// TIA Portal project "2020-11-13_LampeggioMacchinaStati" (V16)
// Programma che gestisce la ventilazione di un motore

(* hardware
DEVICE "Stazione SIMATIC 1200_1"  S71200.Device
   slot 0: "Telaio di montaggio S7-1200"  Rack  V1.0
   slot 1: "PLC_1"  CPU 1215C DC/DC/DC  6ES7 215-1AG40-0XB0  V4.2
*)

// ===== PLC "PLC_1"  CPU 1215C DC/DC/DC =====

VAR_GLOBAL   // PLC tag table "Tabella delle variabili standard"
   "in0_f" AT %I0.0 : Bool;
   "in1_f" AT %I0.1 : Bool;
   "in2_f" AT %I0.2 : Bool;
   "in3_f" AT %I0.3 : Bool;
   "in4_f" AT %I0.4 : Bool;
   "in5_f" AT %I0.5 : Bool;
   "in6_f" AT %I0.6 : Bool;
   "out0" AT %Q0.0 : Bool;
   "out1" AT %Q0.1 : Bool;
   "in7_f" AT %I0.7 : Bool;
   "out2" AT %Q0.2 : Bool;
   "out3" AT %Q0.3 : Bool;
   "out4" AT %Q0.4 : Bool;
   "sempre vero" AT %M7.0 : Bool;   // bit sempre vero
   "uscite byte" AT %QB0 : Byte;   // Uscite fisiche
   "uscite memorie" AT %MB1 : Byte;   // uscite memorie da usare come ingressi
   "out4_M" AT %M1.4 : Bool;
   "out3_M" AT %M1.3 : Bool;
   "out2_M" AT %M1.2 : Bool;
   "out1_M" AT %M1.1 : Bool;
   "out0_M" AT %M1.0 : Bool;
   "ingressi byte" AT %IB0 : Byte;   // Ingressi fisici
   "ingressi memorie" AT %MB0 : Byte;   // Ingressi Na non filtrati
   "in0_na" AT %M0.0 : Bool;
   "in1_na" AT %M0.1 : Bool;
   "in2_na" AT %M0.2 : Bool;
   "in3_na" AT %M0.3 : Bool;
   "in4_na" AT %M0.4 : Bool;
   "in5_na" AT %M0.5 : Bool;
   "in6_na" AT %M0.6 : Bool;
   "in7_na" AT %M0.7 : Bool;
   "out5" AT %Q0.5 : Bool;
   "out6" AT %Q0.6 : Bool;
   "out7" AT %Q0.7 : Bool;
   "out5_M" AT %M1.5 : Bool;
   "out6_M" AT %M1.6 : Bool;
   "out7_M" AT %M1.7 : Bool;
   "ingressi memorie filtrato" AT %MB2 : Byte;
   "in0" AT %M2.0 : Bool;
   "in1" AT %M2.1 : Bool;
   "in2" AT %M2.2 : Bool;
   "in3" AT %M2.3 : Bool;
   "in4" AT %M2.4 : Bool;
   "in5" AT %M2.5 : Bool;
   "in6" AT %M2.6 : Bool;
   "in7" AT %M2.7 : Bool;
   "ingressi memorie_p" AT %MB3 : Byte;
   "in0_p" AT %M3.0 : Bool;   // finecorsa di sicurezza
   "in1_p" AT %M3.1 : Bool;   // presenza tensione al motore
   "in2_p" AT %M3.2 : Bool;   // presenza Allarme
   "in3_p" AT %M3.3 : Bool;   // ventilazione motore ON
   "in4_p" AT %M3.4 : Bool;   // motore troppo caldo
   "in5_p" AT %M3.5 : Bool;   // comando avviamento motore
   "in6_p" AT %M3.6 : Bool;   // comando arresto motore
   "in7_p" AT %M3.7 : Bool;   // Reset memorizzazione Allarme
   "ingressi_memorie_var_p" AT %MB4 : Byte;
   "in0_var_p" AT %M4.0 : Bool;   // finecorsa di sicurezza
   "in1_var_p" AT %M4.1 : Bool;   // presenza tensione al motore
   "in2_var_p" AT %M4.2 : Bool;   // presenza Allarme
   "in3_var_p" AT %M4.3 : Bool;   // ventilazione motore ON
   "in4_var_p" AT %M4.4 : Bool;   // motore troppo caldo
   "in5_var_p" AT %M4.5 : Bool;   // comando avviamento motore
   "in6_var_p" AT %M4.6 : Bool;   // comando arresto motore
   "in7_var_p" AT %M4.7 : Bool;   // Reset memorizzazione Allarme
   "Stato" AT %MB8 : Byte;
   "Stato_futuro" AT %MB9 : Byte;
   "Stato_old" AT %MB10 : Byte;
END_VAR

VAR_GLOBAL CONSTANT   // PLC tag table "Tabella delle variabili standard"
   "maschera NCNA" : Byte := B#2#00000000;   // mettere a 1 i bit NC
   "filtro in0" : Time := T#500ms;
   "filtro in1" : Time := T#100ms;
   "filtro in2" : Time := T#100ms;
   "filtro in3" : Time := T#100ms;
   "filtro in4" : Time := T#100ms;
   "filtro in5" : Time := T#100ms;
   "filtro in6" : Time := T#100ms;
   "filtro in7" : Time := T#100ms;
   "Maschera Out Reset" : Byte := B#2#00000000;
   "Stato_partenza" : Byte := 0;
END_VAR

// folder: System blocks/Program resources

DATA_BLOCK "filtro_in0"   // DB1
{ S7_Optimized_Access := 'TRUE' }
AUTHOR : Simatic
FAMILY : IEC
NAME : IEC_TMR
VERSION : 1.0
// stored: InstanceOfName IEC_TIMER
"IEC_TIMER"
BEGIN
END_DATA_BLOCK

DATA_BLOCK "filtro_in1"   // DB2
{ S7_Optimized_Access := 'TRUE' }
AUTHOR : Simatic
FAMILY : IEC
NAME : IEC_TMR
VERSION : 1.0
// stored: InstanceOfName IEC_TIMER
"IEC_TIMER"
BEGIN
END_DATA_BLOCK

DATA_BLOCK "filtro_in2"   // DB3
{ S7_Optimized_Access := 'TRUE' }
AUTHOR : Simatic
FAMILY : IEC
NAME : IEC_TMR
VERSION : 1.0
// stored: InstanceOfName IEC_TIMER
"IEC_TIMER"
BEGIN
END_DATA_BLOCK

DATA_BLOCK "filtro_in3"   // DB4
{ S7_Optimized_Access := 'TRUE' }
AUTHOR : Simatic
FAMILY : IEC
NAME : IEC_TMR
VERSION : 1.0
// stored: InstanceOfName IEC_TIMER
"IEC_TIMER"
BEGIN
END_DATA_BLOCK

DATA_BLOCK "filtro_in4"   // DB5
{ S7_Optimized_Access := 'TRUE' }
AUTHOR : Simatic
FAMILY : IEC
NAME : IEC_TMR
VERSION : 1.0
// stored: InstanceOfName IEC_TIMER
"IEC_TIMER"
BEGIN
END_DATA_BLOCK

DATA_BLOCK "filtro_in5"   // DB6
{ S7_Optimized_Access := 'TRUE' }
AUTHOR : Simatic
FAMILY : IEC
NAME : IEC_TMR
VERSION : 1.0
// stored: InstanceOfName IEC_TIMER
"IEC_TIMER"
BEGIN
END_DATA_BLOCK

DATA_BLOCK "filtro_in6"   // DB7
{ S7_Optimized_Access := 'TRUE' }
AUTHOR : Simatic
FAMILY : IEC
NAME : IEC_TMR
VERSION : 1.0
// stored: InstanceOfName IEC_TIMER
"IEC_TIMER"
BEGIN
END_DATA_BLOCK

DATA_BLOCK "filtro_in7"   // DB8
{ S7_Optimized_Access := 'TRUE' }
AUTHOR : Simatic
FAMILY : IEC
NAME : IEC_TMR
VERSION : 1.0
// stored: InstanceOfName IEC_TIMER
"IEC_TIMER"
BEGIN
END_DATA_BLOCK

// folder: (top level)

FUNCTION "Ingressi e uscite" : Void   // FC1, LAD
{ S7_Optimized_Access := 'TRUE' }
VERSION : 0.1
   VAR_TEMP   // added for the SCL form of the ladder/FBD networks
      _w1 : Bool;
   END_VAR
BEGIN

REGION Network 1: creazione immagine uscite (MB1) da usare come ingressi
   // creazione immagine uscite (MB1) da usare come ingressi
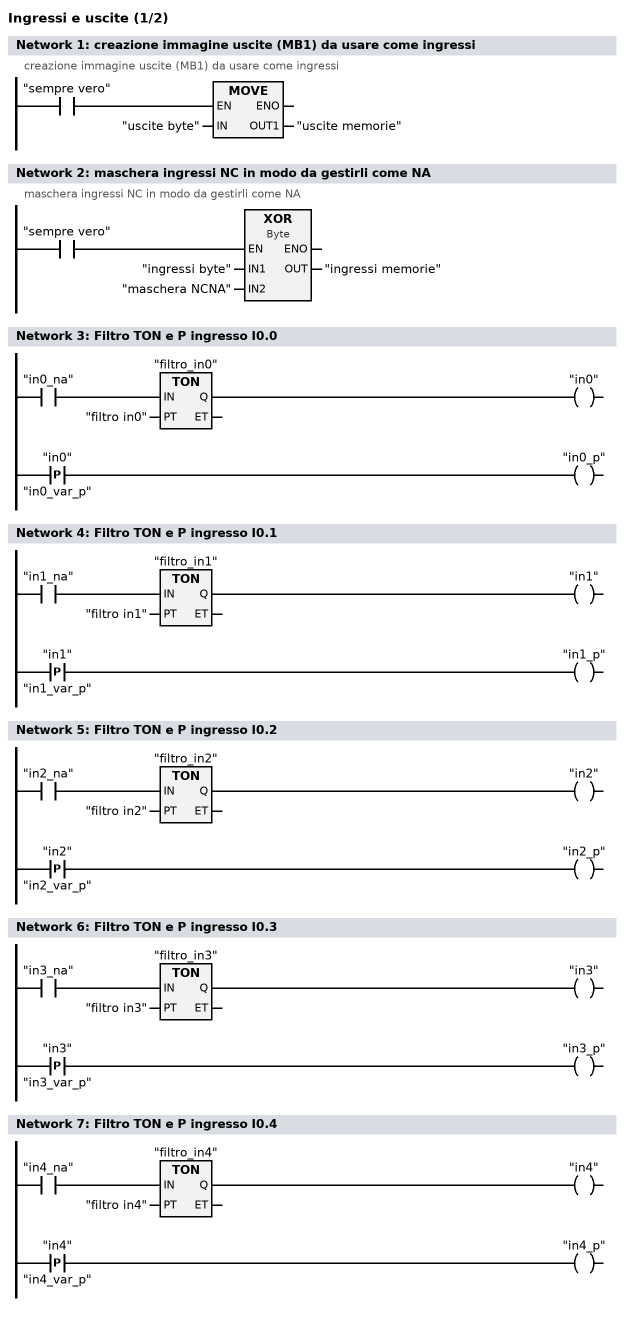
   RUNG wire#powerrail
      Contact( "sempre vero" )
      { S7_GenerateENO := "TRUE" } Move(in := "uscite byte", out1 => "uscite memorie")
   END_RUNG
   // the same network as SCL:
   IF "sempre vero" THEN "uscite memorie" := "uscite byte"; END_IF;
END_REGION

REGION Network 2: maschera ingressi NC in modo da gestirli come NA
   // maschera ingressi NC in modo da gestirli come NA
   IF "sempre vero" THEN "ingressi memorie" := "ingressi byte" XOR "maschera NCNA"; END_IF;
END_REGION

REGION Network 3: Filtro TON e P ingresso I0.0
   "filtro_in0".TON(IN := "in0_na", PT := "filtro in0");
   "in0" := "filtro_in0".Q;
   #_w1 := "in0" AND NOT "in0_var_p";   // rising edge of "in0"
   "in0_var_p" := "in0";
   "in0_p" := #_w1;
END_REGION

REGION Network 4: Filtro TON e P ingresso I0.1
   "filtro_in1".TON(IN := "in1_na", PT := "filtro in1");
   "in1" := "filtro_in1".Q;
   #_w1 := "in1" AND NOT "in1_var_p";   // rising edge of "in1"
   "in1_var_p" := "in1";
   "in1_p" := #_w1;
END_REGION

REGION Network 5: Filtro TON e P ingresso I0.2
   "filtro_in2".TON(IN := "in2_na", PT := "filtro in2");
   "in2" := "filtro_in2".Q;
   #_w1 := "in2" AND NOT "in2_var_p";   // rising edge of "in2"
   "in2_var_p" := "in2";
   "in2_p" := #_w1;
END_REGION

REGION Network 6: Filtro TON e P ingresso I0.3
   "filtro_in3".TON(IN := "in3_na", PT := "filtro in3");
   "in3" := "filtro_in3".Q;
   #_w1 := "in3" AND NOT "in3_var_p";   // rising edge of "in3"
   "in3_var_p" := "in3";
   "in3_p" := #_w1;
END_REGION

REGION Network 7: Filtro TON e P ingresso I0.4
   "filtro_in4".TON(IN := "in4_na", PT := "filtro in4");
   "in4" := "filtro_in4".Q;
   #_w1 := "in4" AND NOT "in4_var_p";   // rising edge of "in4"
   "in4_var_p" := "in4";
   "in4_p" := #_w1;
END_REGION

REGION Network 8: Filtro TON e P ingresso I0.5
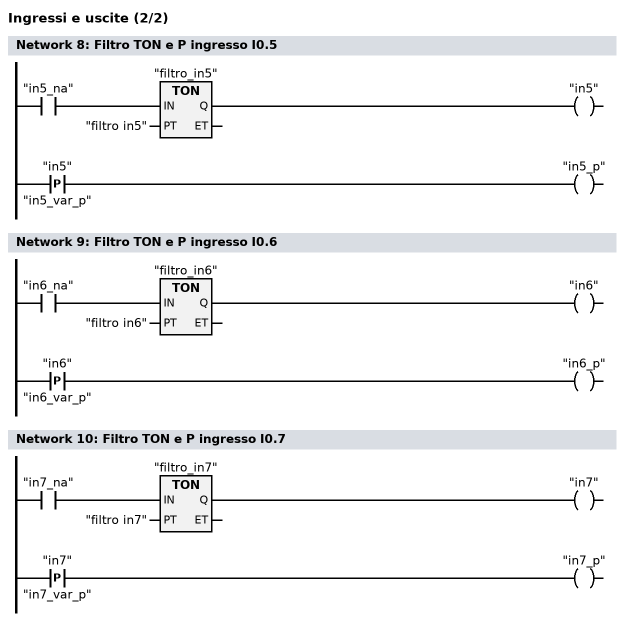
   "filtro_in5".TON(IN := "in5_na", PT := "filtro in5");
   "in5" := "filtro_in5".Q;
   #_w1 := "in5" AND NOT "in5_var_p";   // rising edge of "in5"
   "in5_var_p" := "in5";
   "in5_p" := #_w1;
END_REGION

REGION Network 9: Filtro TON e P ingresso I0.6
   "filtro_in6".TON(IN := "in6_na", PT := "filtro in6");
   "in6" := "filtro_in6".Q;
   #_w1 := "in6" AND NOT "in6_var_p";   // rising edge of "in6"
   "in6_var_p" := "in6";
   "in6_p" := #_w1;
END_REGION

REGION Network 10: Filtro TON e P ingresso I0.7
   "filtro_in7".TON(IN := "in7_na", PT := "filtro in7");
   "in7" := "filtro_in7".Q;
   #_w1 := "in7" AND NOT "in7_var_p";   // rising edge of "in7"
   "in7_var_p" := "in7";
   "in7_p" := #_w1;
END_REGION
END_FUNCTION

ORGANIZATION_BLOCK "Main"   // OB1, LAD, ProgramCycle
TITLE = "Main Program Sweep (Cycle)"
{ S7_Optimized_Access := 'TRUE' }
VERSION : 0.1
// Base per macchina a stati
// 1) disegnare macchina a stati
// 2) in analogia con il programma base, configurare costanti (mascheraNANC, filtri, eventuali tempi della sequenza) e variabili  (Q0.x, M1.x, M2.x e, se serve, M3.x) ATTENZIONE! Mettere tutte le nuove variabili a partire dall'indirizzo 12, lasciando inalterata la mappatura da 0 a 10
// 3) elencare passi a partire dal segmento 5, rimuovendo gli esempi, e impostando solo il commento in visualizzazione compatta 
// 4) elencare transizioni condizionate a partire dal segmento 2 (priorità all'ultimo segmento) rimuovendo gli esempi e impostando solo il commento in visualizzazione compatta 
// 5) elencare transizioni incondizionate a seguire di quelle condizionate, rimuovendo gli esempi,  e impostando solo il commento in visualizzazione compatta 
// 6) implementare passi secondo il commento
// 7) implementare transizioni condizionate e incondizionate seguendo il commento
// 8) lasciare inalterato il segmento del passaggio di stato (da stato_futuro a stato)
// 9) controllare compattando/espandendo i segmenti e guardando i timer in blocchi di sistema/risorse del programma 
// 10) compilare, caricare e testare
// NOTA: inserire eventuali Function o istruzioni comuni a tutti gli stati a seguire del segmento 1, subito prima delle transizioni
BEGIN

REGION Network 1: richiamo FC
   // creazione immagine uscite (MB1) da usare come ingressi
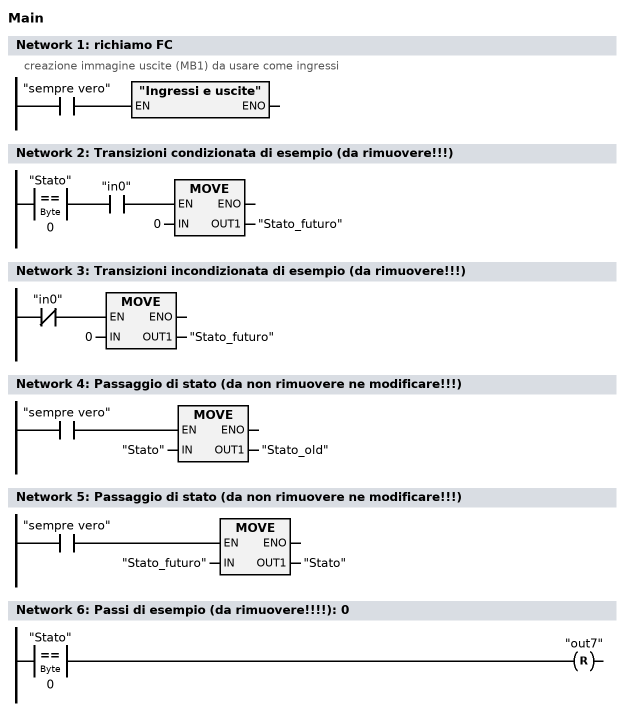
   RUNG wire#powerrail
      Contact( "sempre vero" )
      "Ingressi e uscite"()
   END_RUNG
   // the same network as SCL:
   IF "sempre vero" THEN "Ingressi e uscite"(); END_IF;
END_REGION

REGION Network 2: Transizioni condizionata di esempio (da rimuovere!!!)
   RUNG wire#powerrail
      { S7_Templates := "SrcType := Byte" } EQ_Contact(in1 := "Stato", in2 := 0)
      Contact( "in0" )
      { S7_GenerateENO := "TRUE" } Move(in := 0, out1 => "Stato_futuro")
   END_RUNG
   // the same network as SCL:
   IF ("Stato" = 0) AND "in0" THEN "Stato_futuro" := 0; END_IF;
END_REGION

REGION Network 3: Transizioni incondizionata di esempio (da rimuovere!!!)
   RUNG wire#powerrail
      I_Contact( "in0" )
      { S7_GenerateENO := "TRUE" } Move(in := 0, out1 => "Stato_futuro")
   END_RUNG
   // the same network as SCL:
   IF NOT "in0" THEN "Stato_futuro" := 0; END_IF;
END_REGION

REGION Network 4: Passaggio di stato (da non rimuovere ne modificare!!!)
   RUNG wire#powerrail
      Contact( "sempre vero" )
      { S7_GenerateENO := "TRUE" } Move(in := "Stato", out1 => "Stato_old")
   END_RUNG
   // the same network as SCL:
   IF "sempre vero" THEN "Stato_old" := "Stato"; END_IF;
END_REGION

REGION Network 5: Passaggio di stato (da non rimuovere ne modificare!!!)
   RUNG wire#powerrail
      Contact( "sempre vero" )
      { S7_GenerateENO := "TRUE" } Move(in := "Stato_futuro", out1 => "Stato")
   END_RUNG
   // the same network as SCL:
   IF "sempre vero" THEN "Stato" := "Stato_futuro"; END_IF;
END_REGION

REGION Network 6: Passi di esempio (da rimuovere!!!!): 0
   RUNG wire#powerrail
      { S7_Templates := "SrcType := Byte" } EQ_Contact(in1 := "Stato", in2 := 0)
      R_Coil( "out7" )
   END_RUNG
   // the same network as SCL:
   IF "Stato" = 0 THEN "out7" := FALSE; END_IF;
END_REGION
END_ORGANIZATION_BLOCK

ORGANIZATION_BLOCK "Startup"   // OB100, LAD, Startup
TITLE = "Complete Restart"
{ S7_Optimized_Access := 'TRUE' }
VERSION : 0.1
   VAR_INPUT
      LostRetentive : Bool;   // True if retentive data are lost
      LostRTC : Bool;   // True if real time clock is lost
   END_VAR
BEGIN

REGION Network 1: bit sempre vero
   // creazione bit sempre vero
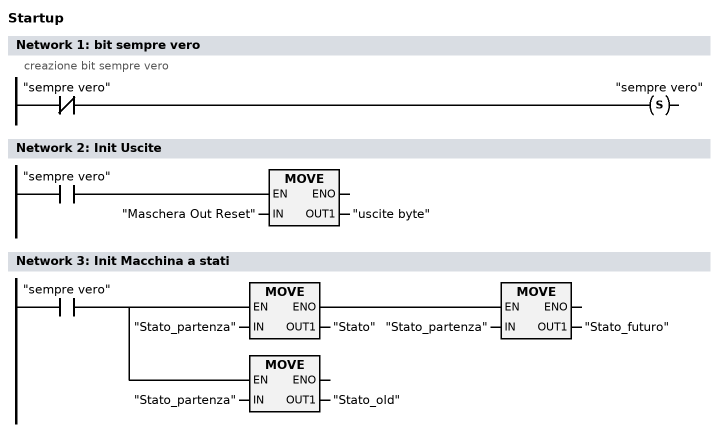
   RUNG wire#powerrail
      I_Contact( "sempre vero" )
      S_Coil( "sempre vero" )
   END_RUNG
   // the same network as SCL:
   IF NOT "sempre vero" THEN "sempre vero" := TRUE; END_IF;
END_REGION

REGION Network 2: Init Uscite
   RUNG wire#powerrail
      Contact( "sempre vero" )
      { S7_GenerateENO := "TRUE" } Move(in := "Maschera Out Reset", out1 => "uscite byte")
   END_RUNG
   // the same network as SCL:
   IF "sempre vero" THEN "uscite byte" := "Maschera Out Reset"; END_IF;
END_REGION

REGION Network 3: Init Macchina a stati
   RUNG wire#powerrail
      Contact( "sempre vero" )
      wire#w1
      { S7_GenerateENO := "TRUE" } Move(in := "Stato_partenza", out1 => "Stato")
      { S7_GenerateENO := "TRUE" } Move(in := "Stato_partenza", out1 => "Stato_futuro")
   END_RUNG
   RUNG wire#w1
      Move(in := "Stato_partenza", out1 => "Stato_old")
   END_RUNG
   // the same network as SCL:
   // ENO of a box is taken as its EN; it also drops when the box reports an error
   IF "sempre vero" THEN
       "Stato" := "Stato_partenza";
       "Stato_futuro" := "Stato_partenza";
       "Stato_old" := "Stato_partenza";
   END_IF;
END_REGION
END_ORGANIZATION_BLOCK